// TIA Portal V15.1 export
FUNCTION_BLOCK "MotorControl"   // FB
AUTHOR : Pat
// Controls a motor with start/stop logic
BEGIN
END_FUNCTION_BLOCK
